// TIA Portal V19 export
VAR_GLOBAL   // PLC tag table "TT - System"
   System_Byte AT %MB254 : Byte;
   FirstScan AT %M254.0 : Bool;
   DiagStatusUpdate AT %M254.1 : Bool;
   AlwaysTRUE AT %M254.2 : Bool;
   AlwaysFALSE AT %M254.3 : Bool;
END_VAR
